{attribute 'pack_mode' := '1'}
TYPE TVisionPartData :
	STRUCT
		lrX				: LREAL;
		lrY				: LREAL;
		lrTheta			: LREAL;
		lrScore			: LREAL;
		bValid			: BOOL;
		bPresent			: BOOL;
		bImageGrabbed	: BOOL;
	END_STRUCT
END_TYPE

(* stored: Version 1.1.0.1, ProductVersion 3.1.4022.12
   DUT TVisionPartData: Id {60b7070f-cea5-4ff7-afee-c0461561b203} *)
